Xinje XDPPro project, PLC1: XD5-48T6 (software 3.5.3 2018-11-19)

PROGRAM Ladder

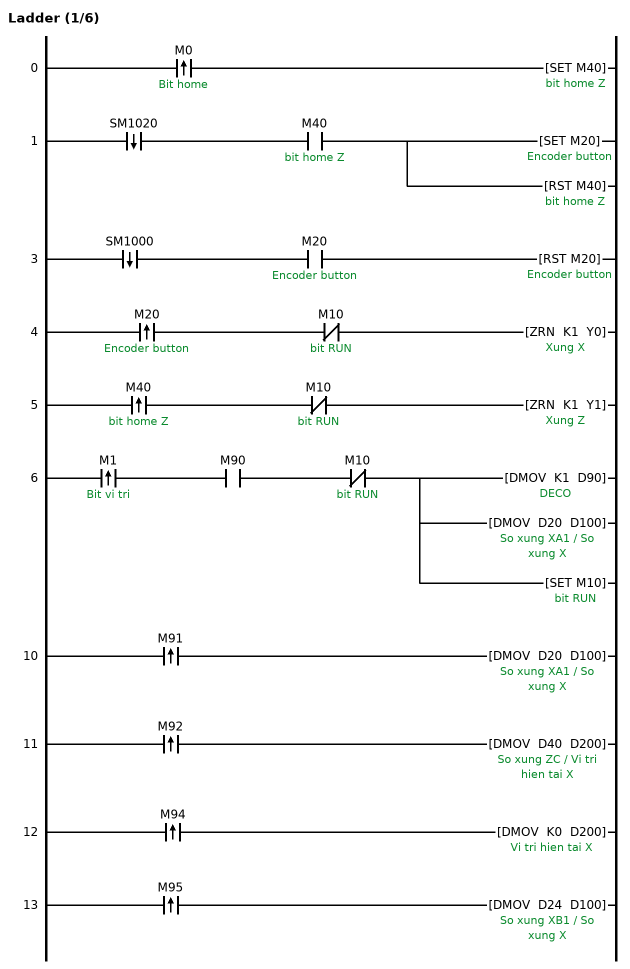
LDP    M0	; Bit home
SET    M40	; bit home Z
LDF    SM1020
AND    M40	; bit home Z
SET    M20	; Encoder button
RST    M40	; bit home Z
LDF    SM1000
AND    M20	; Encoder button
RST    M20	; Encoder button
LDP    M20	; Encoder button
ANI    M10	; bit RUN
ZRN    K1 Y0	; Xung X
LDP    M40	; bit home Z
ANI    M10	; bit RUN
ZRN    K1 Y1	; Xung Z
LDP    M1	; Bit vi tri
AND    M90
ANI    M10	; bit RUN
DMOV   K1 D90	; DECO
DMOV   D20 D100	; So xung XA1 / So xung X
SET    M10	; bit RUN
LDP    M91
DMOV   D20 D100	; So xung XA1 / So xung X
LDP    M92
DMOV   D40 D200	; So xung ZC / Vi tri hien tai X
LDP    M94
DMOV   K0 D200	; Vi tri hien tai X
LDP    M95
DMOV   D24 D100	; So xung XB1 / So xung X

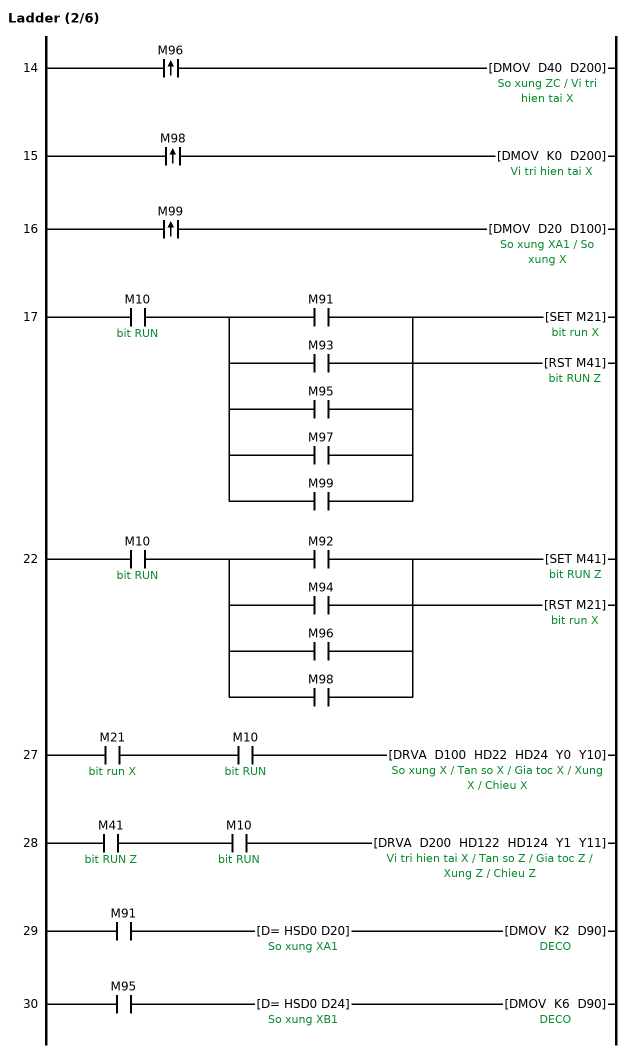
LDP    M96
DMOV   D40 D200	; So xung ZC / Vi tri hien tai X
LDP    M98
DMOV   K0 D200	; Vi tri hien tai X
LDP    M99
DMOV   D20 D100	; So xung XA1 / So xung X
LD     M10	; bit RUN
LD     M91
OR     M93
OR     M95
OR     M97
OR     M99
ANB
SET    M21	; bit run X
RST    M41	; bit RUN Z
LD     M10	; bit RUN
LD     M92
OR     M94
OR     M96
OR     M98
ANB
SET    M41	; bit RUN Z
RST    M21	; bit run X
LD     M21	; bit run X
AND    M10	; bit RUN
DRVA   D100 HD22 HD24 Y0 Y10	; So xung X / Tan so X / Gia toc X / Xung X / Chieu X
LD     M41	; bit RUN Z
AND    M10	; bit RUN
DRVA   D200 HD122 HD124 Y1 Y11	; Vi tri hien tai X / Tan so Z / Gia toc Z / Xung Z / Chieu Z
LD     M91
DAND=  HSD0 D20	; So xung XA1
DMOV   K2 D90	; DECO
LD     M95
DAND=  HSD0 D24	; So xung XB1
DMOV   K6 D90	; DECO

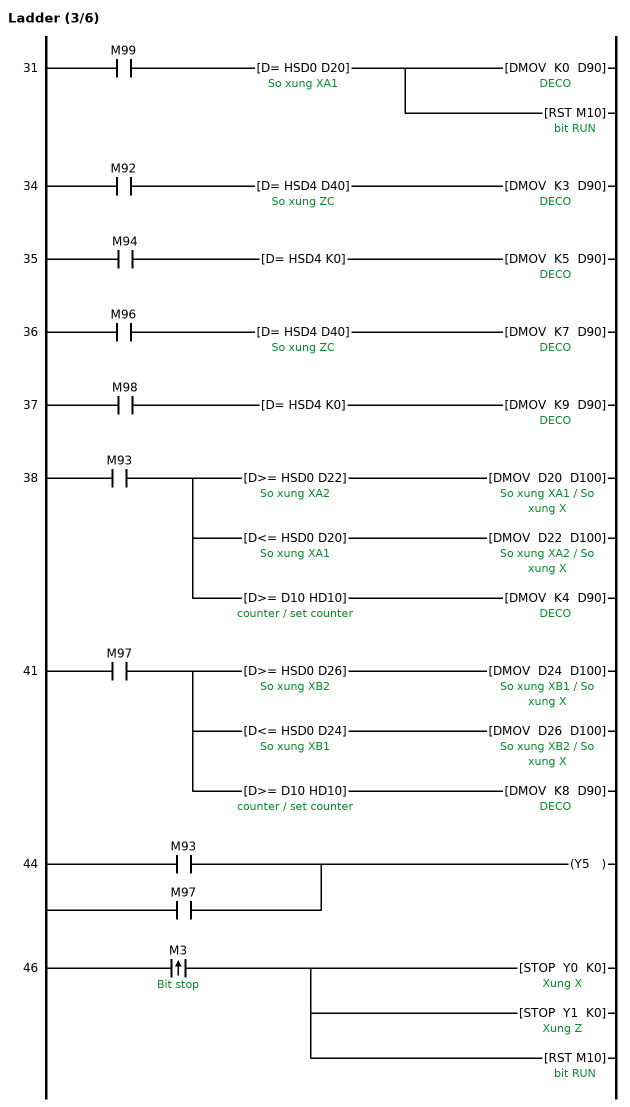
LD     M99
DAND=  HSD0 D20	; So xung XA1
DMOV   K0 D90	; DECO
RST    M10	; bit RUN
LD     M92
DAND=  HSD4 D40	; So xung ZC
DMOV   K3 D90	; DECO
LD     M94
DAND=  HSD4 K0
DMOV   K5 D90	; DECO
LD     M96
DAND=  HSD4 D40	; So xung ZC
DMOV   K7 D90	; DECO
LD     M98
DAND=  HSD4 K0
DMOV   K9 D90	; DECO
LD     M93
MPS
DAND>= HSD0 D22	; So xung XA2
DMOV   D20 D100	; So xung XA1 / So xung X
MRD
DAND<= HSD0 D20	; So xung XA1
DMOV   D22 D100	; So xung XA2 / So xung X
MPP
DAND>= D10 HD10	; counter / set counter
DMOV   K4 D90	; DECO
LD     M97
MPS
DAND>= HSD0 D26	; So xung XB2
DMOV   D24 D100	; So xung XB1 / So xung X
MRD
DAND<= HSD0 D24	; So xung XB1
DMOV   D26 D100	; So xung XB2 / So xung X
MPP
DAND>= D10 HD10	; counter / set counter
DMOV   K8 D90	; DECO
LD     M93
OR     M97
OUT    Y5
LDP    M3	; Bit stop
STOP   Y0 K0	; Xung X
STOP   Y1 K0	; Xung Z
RST    M10	; bit RUN

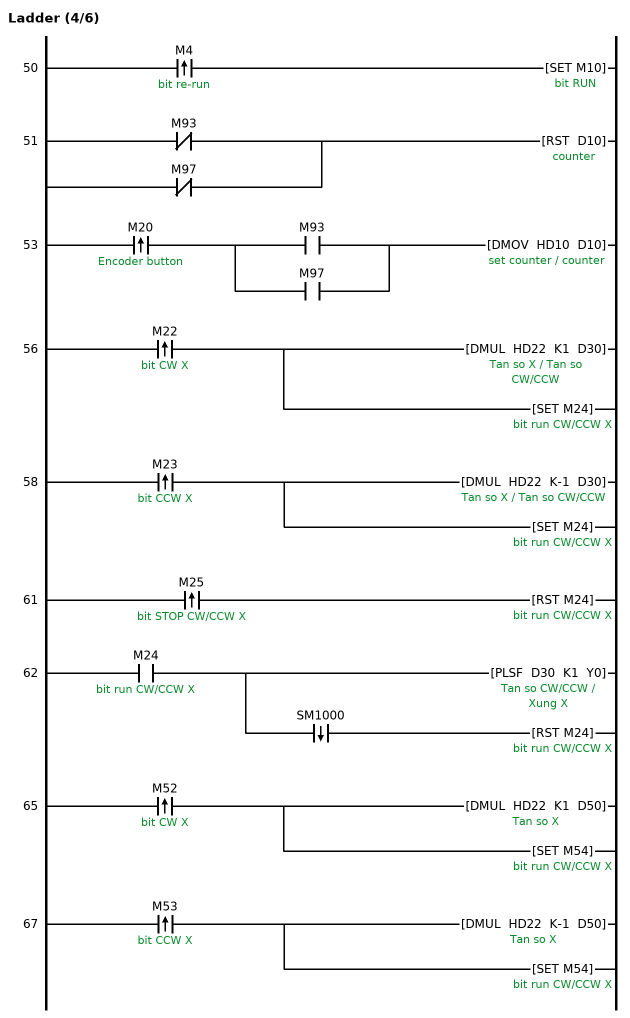
LDP    M4	; bit re-run
SET    M10	; bit RUN
LDI    M93
ORI    M97
RST    D10	; counter
LDP    M20	; Encoder button
LD     M93
OR     M97
ANB
DMOV   HD10 D10	; set counter / counter
LDP    M22	; bit CW X
DMUL   HD22 K1 D30	; Tan so X / Tan so CW/CCW
SET    M24	; bit run CW/CCW X
LDP    M23	; bit CCW X
DMUL   HD22 K-1 D30	; Tan so X / Tan so CW/CCW
SET    M24	; bit run CW/CCW X
LDP    M25	; bit STOP CW/CCW X
RST    M24	; bit run CW/CCW X
LD     M24	; bit run CW/CCW X
PLSF   D30 K1 Y0	; Tan so CW/CCW / Xung X
ANDF   SM1000
RST    M24	; bit run CW/CCW X
LDP    M52	; bit CW X
DMUL   HD22 K1 D50	; Tan so X
SET    M54	; bit run CW/CCW X
LDP    M53	; bit CCW X
DMUL   HD22 K-1 D50	; Tan so X
SET    M54	; bit run CW/CCW X

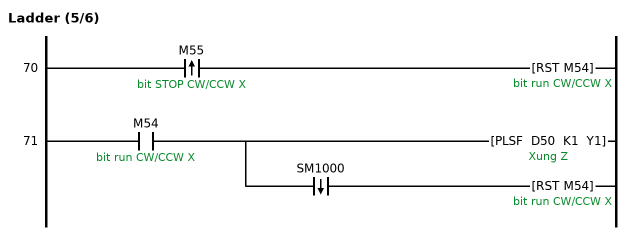
LDP    M55	; bit STOP CW/CCW X
RST    M54	; bit run CW/CCW X
LD     M54	; bit run CW/CCW X
PLSF   D50 K1 Y1	; Xung Z
ANDF   SM1000
RST    M54	; bit run CW/CCW X

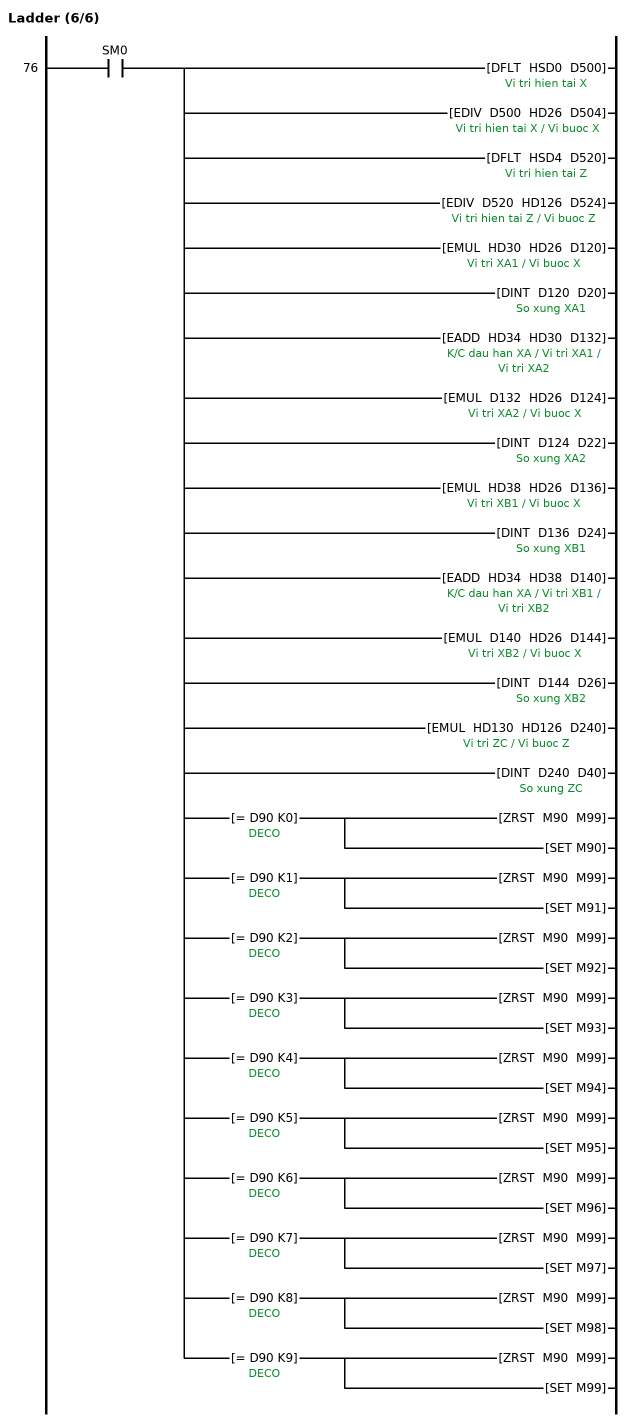
LD     SM0
DFLT   HSD0 D500	; Vi tri hien tai X
EDIV   D500 HD26 D504	; Vi tri hien tai X / Vi buoc X
DFLT   HSD4 D520	; Vi tri hien tai Z
EDIV   D520 HD126 D524	; Vi tri hien tai Z / Vi buoc Z
EMUL   HD30 HD26 D120	; Vi tri XA1 / Vi buoc X
DINT   D120 D20	; So xung XA1
EADD   HD34 HD30 D132	; K/C dau han XA / Vi tri XA1 / Vi tri XA2
EMUL   D132 HD26 D124	; Vi tri XA2 / Vi buoc X
DINT   D124 D22	; So xung XA2
EMUL   HD38 HD26 D136	; Vi tri XB1 / Vi buoc X
DINT   D136 D24	; So xung XB1
EADD   HD34 HD38 D140	; K/C dau han XA / Vi tri XB1 / Vi tri XB2
EMUL   D140 HD26 D144	; Vi tri XB2 / Vi buoc X
DINT   D144 D26	; So xung XB2
EMUL   HD130 HD126 D240	; Vi tri ZC / Vi buoc Z
DINT   D240 D40	; So xung ZC
MPS
AND=   D90 K0	; DECO
ZRST   M90 M99
SET    M90
MRD
AND=   D90 K1	; DECO
ZRST   M90 M99
SET    M91
MRD
AND=   D90 K2	; DECO
ZRST   M90 M99
SET    M92
MRD
AND=   D90 K3	; DECO
ZRST   M90 M99
SET    M93
MRD
AND=   D90 K4	; DECO
ZRST   M90 M99
SET    M94
MRD
AND=   D90 K5	; DECO
ZRST   M90 M99
SET    M95
MRD
AND=   D90 K6	; DECO
ZRST   M90 M99
SET    M96
MRD
AND=   D90 K7	; DECO
ZRST   M90 M99
SET    M97
MRD
AND=   D90 K8	; DECO
ZRST   M90 M99
SET    M98
MPP
AND=   D90 K9	; DECO
ZRST   M90 M99
SET    M99